PROGRAM MAIN
VAR
END_VAR

END_PROGRAM

(* stored: Version 1.1.0.1
   POU MAIN: Id {435e48f9-95ac-4610-a340-790913c8bea3} *)
